TYPE ENUM_StepperMotorState :
(
	LAS_Stepper_Uninitialized := 0,
    LAS_Stepper_Moving := 2,
    LAS_Stepper_Idle := 3,
    LAS_Stepper_Error := 6,
	LAS_Stepper_FastPass := 1,
	LAS_Stepper_SlowPass := 4,
	LAS_Stepper_WaitingForTrigger := 5,
	LAS_Stepper_Hardware_Check := 7
);
END_TYPE

(* stored: Version 1.1.0.1, ProductVersion 3.1.4026.11
   DUT ENUM_StepperMotorState: Id {0ba129ba-95f5-4579-9013-1d3c3672a9df} *)
